// TIA Portal V16 export
// export: Created 2021-09-08T12:44:32.5996252Z, ExportSetting WithDefaults, DisplayName Totally Integrated Automation Portal, DisplayVersion V16 Update 3, DisplayName TIA Portal Version Control Interface, DisplayVersion V16 Update 2, DisplayName TIA Portal Openness, DisplayVersion V16 Update 3, DisplayName TIA Portal Teamcenter Gateway, DisplayVersion V16, DisplayName STEP 7 Professional, DisplayVersion V16 Update 3, DisplayName STEP 7 Safety, DisplayVersion V16, DisplayName WinCC Advanced, DisplayVersion V16 Update 3
VAR_GLOBAL   // PLC tag table "A10_AI"
   aiLT201 AT %IW68 : Int;   // Рівень ємності TW201 LT201
   aiLT202 AT %IW70 : Int;   // Рівень ємності TW202 LT202
   aiPT301 AT %IW72 : Int;   // Тиск PS3 PT301
   aiPT401 AT %IW74 : Int;   // Тиск MDF4 PT401
   aiPT501 AT %IW76 : Int;   // Тиск повітря UF PT501
   aiPT502 AT %IW78 : Int;   // Тиск вхідної води UF PT502
   aiPT503 AT %IW80 : Int;   // Тиск фільтрата UF PT503
   aiPT504 AT %IW82 : Int;   // Тиск стічних вод UF PT504
   aiPT505 AT %IW84 : Int;   // Тиск вхідної води UF PT505
   aiPT506 AT %IW86 : Int;   // Тиск фільтрата UF PT506
   aiPT507 AT %IW88 : Int;   // Тиск стічних вод UF PT507
   aiLT601 AT %IW90 : Int;   // Рівень ємності TW601 LT601
   aiPT701 AT %IW92 : Int;   // Тиск PS7 PT701
   aiPT901 AT %IW94 : Int;   // Тиск насоса RO PT901
   aiPT902 AT %IW96 : Int;   // Тиск концентрата RO PT902
   aiLT1101 AT %IW98 : Int;   // Рівень ємності TW1101 LT1101
   aiPT1201 AT %IW100 : Int;   // Тиск PS12 PT1201
   aiPT1301 AT %IW102 : Int;   // Тиск насоса NF PT1301
   aiPT1302 AT %IW104 : Int;   // Тиск концентрата NF PT1302
   aiLT1401 AT %IW106 : Int;   // Рівень ємності TW1401 LT1401
   aiLT1402 AT %IW108 : Int;   // Рівень ємності TW1402 LT1402
   aiPT1501 AT %IW110 : Int;   // Тиск PS15 PT1501
   aiPT1701 AT %IW112 : Int;   // Тиск MCF17 PT1701
   aiLT1801 AT %IW114 : Int;   // Рівень ємності TW1801 LT1801
   aiFM501 AT %IW116 : Int;   // Витрата вхідної води UF FM501
   aiFM502 AT %IW118 : Int;   // Витрата вхідної води UF FM502
   aiFM901 AT %IW120 : Int;   // Витрата пермеату RO FM901
   aiFM902 AT %IW122 : Int;   // Витрата концентрату RO FM902
   aiFM1301 AT %IW124 : Int;   // Витрата пермеату NF FM901
   aiFM1302 AT %IW126 : Int;   // Витрата концентрату NF FM902
   aiORP801 AT %IW128 : Int;   // ORP води на UF ORP801
   aiCDI901 AT %IW130 : Int;   // Електропровідність пермеату RO CDI901
   aiCDI1301 AT %IW132 : Int;   // Електропровідність пермеату RO CD1301
   aiCDI1302 AT %IW134 : Int;   // Електропровідність після змішування CD1302
   aiCDI1801 AT %IW136 : Int;   // Електропровідність стічних вод CD1801
   PIW74_Reserve AT %IW138 : Int;   // Резерв
   PIW76_Reserve AT %IW140 : Int;   // Резерв
   PIW78_Reserve AT %IW142 : Int;   // Резерв
   PIW80_Reserve AT %IW144 : Int;   // Резерв
   PIW82_Reserve AT %IW146 : Int;   // Резерв
END_VAR
VAR_GLOBAL CONSTANT   // user constants
   iwLT201 : Int := 0;
   iwLT202 : Int := 1;
   iwPT301 : Int := 2;
   iwPT401 : Int := 3;
   iwPT501 : Int := 4;
   iwPT502 : Int := 5;
   iwPT503 : Int := 6;
   iwPT504 : Int := 7;
   iwPT505 : Int := 8;
   iwPT506 : Int := 9;
   iwPT507 : Int := 10;
   iwLT601 : Int := 11;
   iwPT701 : Int := 12;
   iwPT901 : Int := 13;
   iwPT902 : Int := 14;
   iwLT1101 : Int := 15;
   iwPT1201 : Int := 16;
   iwPT1301 : Int := 17;
   iwPT1302 : Int := 18;
   iwLT1401 : Int := 19;
   iwLT1402 : Int := 20;
   iwPT1501 : Int := 21;
   iwPT1701 : Int := 22;
   iwLT1801 : Int := 23;
   iwFM501 : Int := 24;
   iwFM502 : Int := 25;
   iwFM901 : Int := 26;
   iwFM902 : Int := 27;
   iwFM1301 : Int := 28;
   iwFM1302 : Int := 29;
   iwORP801 : Int := 30;
   iwCDI901 : Int := 31;
   iwCDI1301 : Int := 32;
   iwCDI1302 : Int := 33;
   iwCDI1801 : Int := 34;
   iw74_Reserve : Int := 35;
   iw76_Reserve : Int := 36;
   iw78_Reserve : Int := 37;
   iw80_Reserve : Int := 38;
   iw82_Reserve : Int := 39;
END_VAR
